// SIMATIC S7-200 project (STEP 7-Micro/WIN), CPU 226 REL 01.22

SYMBOL_TABLE USR1
First_Scan_On    SM0.1    // This bit is on for the first scan cycle only.
END_SYMBOL_TABLE

ORGANIZATION_BLOCK MAIN:OB1
TITLE=At system startup, during the first scan cycle, the first scan flag is set, enabling all interrupt events and setting the message enable flag to ensure that runtime information can be displayed. Since interrupts need to be enabled after the system stabilizes, the falling edge of the first scan flag triggers after the first scan, attaching the interrupt event to the interrupt.
// When the external timer feedback signal is OFF, indicating that the external timer is idle, the system sets the timer start signal and subsequently activates the internal timer. Only when the external timer feedback signal is OFF will the timer start signal be set, ensuring that the external timer starts operating in the correct state. The internal timer has a preset time of 32 seconds and begins counting, while the external timer is configured by the user, with its feedback signal designed to return within the 32-second window.
// The external timer sends the feedback signal after its configured duration, and its rising edge triggers the interrupt. The system design requires that the rising edge of the feedback signal triggers the interrupt during the counting period of the internal timer to meet measurement accuracy. During interrupt handling, if the timer start signal is set, the system copies the current value of the internal timer to the measurement value and displays it for operator monitoring. Since display accuracy is critical, the measurement value precisely copies the value of the internal timer at the moment of interruption. Subsequently, the system resets the timer start signal and detaches the interrupt event, preparing for the next measurement.
BEGIN
Network 1 //  Enable Interrupts and Enable TD 200 Message
//  Load special memory bit SM0.1 to process this network in the
//  first scan cycle only.
//  Enable all interrupt events.
//  Set variable memory bit V12.7 to enable the message on the
//  TD 200.
// 
LD     First_Scan_On:SM0.1   // Load SM0.1.
ENI                          // Enable all interrupt events.
S      V12.7, 1              // Set V12.7 to enable TD 200
// message.
Network 2 //  Attach Interrupt Routine and Set Output Signal
//  Load input I0.0 as a Normally Closed contact to enable power flow
//  if the input is not set.
//  Handle special memory bit SM0.1 as a Normally Closed contact to
//  enable power flow if the bit is not set, that is, during every
//  scan cycle except the first.
//  After the first scan cycle is complete, the on-to-off transition
//  at special memory bit SM0.1 (Normally Closed contact) creates a
//  positive transition (Edge Up). This positive transition causes
//  the program to attach interrupt event 0 to the interrupt routine
//  INT5. Interrupt event 0 is triggered every time there is a positive
//  transition at input I0.0. After the second scan cycle, the
//  on-to-off transition at input I0.0 enables power flow to this
//  network.
//  Set output Q0.0 immediately. The power flow at output Q0.0 enables
//  the internal timer T32, moves the value in T32 to variable memory
//  word VW117 for display on the TD 200, and then resets Q0.0 to
//  restart both the internal and external timers.
// 
LDN    I0.0                  // Load input I0.0 as a Normally
// Closed contact.
AN     First_Scan_On:SM0.1   // If there is no power flow at
// SM0.1 (not first scan cycle)
EU                           // and there is a positive transition
// (on-to-off),
ATCH   INT_5:INT5, 0         // attach interrupt event 0 to
// INT5 and
SI     Q0.0, 1               // set output Q0.0 immediately.
Network 3 //  Turn on Timer T32
//  Load output Q0.0.
//  If output Q0.0 is set,
//  enable timer T32 with a Preset Time (PT) of 32000. Timer T32 has
//  a resolution of 1 ms. A PT of 32000 is therefore equal to 32 s.
// 
LD     Q0.0                  // Load output Q0.0.
// If output Q0.0 is set,
TON    T32, +32000           // enable timer T32 with a PT
// of 32000 (32 s).
Network 4 //  Main Program End
//  End the main program.
// MEND					// End the main program.
// 
// ***INTERRUPT ROUTINE***
// 
// 
Network 5 //  Interrupt Routine INT5
//  Start INT5.
// 
END_ORGANIZATION_BLOCK

INTERRUPT_BLOCK INT_5:INT5
TITLE=
BEGIN
Network 2 //  Copy Time Value to TD 200 Display and Restart Timer
//  Load output Q0.0.
//  If output Q0.0 is set,
//  move the time value in timer T32 to variable memory word VW115
//  to display the number on the TD 200.
//  Reset output Q0.0 (this will clear the value in timer T32).
//  Detach interrupt event 0 from INT5.
// 
LD     Q0.0                  // Load output Q0.0.
// If output Q0.0 is set,
MOVW   T32, VW115            // move the value in T32 to
// variable memory word VW115.
R      Q0.0, 1               // reset output bit Q0.0, and
DTCH   0                     // detach interrupt event 0 from
// INT5.
Network 3 //  End of Interrupt Routine INT5
//  End INT5.
// RETI					// End INT5.
// 
END_INTERRUPT_BLOCK

DATA_BLOCK_TAB USER1
BEGIN
//Data Block DB1 (V Memory):
// BEGIN TD200_BLOCK 0
// (Comments within this block should not be edited or removed)
VB0      'TD'                // TD 200 Identification
VB2      16#10               // Set Language to English, set Update to As fast as possible
VB3      16#0                // Set the display to 20 character mode; Up key V3.2; Down key V3.3
VB4      1                   // Set the number of messages
VB5      0                   // Set the Function Keys notification bits to M0.0 - M0.7 
VW6      100                 // Set the starting address for messages to VW100
VW8      12                  // Set the starting address for message enable bits to VW12
// MESSAGE 1
// Message Enable Bit V12.7
VB100    ' POT Value:  '
VB113    16#10               // Edit Notification V113.2; No Acknowledgement; No Password;
VB114    16#33               // Unsigned Word;  3 Digits to the right of the decimal;
VW115    16#0                // Embedded Data Value: Move data for display here.
VB117    '   '
// END TD200_BLOCK 0
END_DATA_BLOCK_TAB
